FUNCTION_BLOCK Stage11 (* Template for a Basic Function Block Type *)
  (* Standard: 61499-2 *)
  (* Version 1.0, 2021-06-20, HP *)
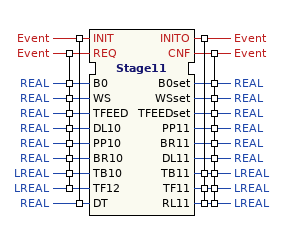
  EVENT_INPUT
    INIT WITH DT; (* Initialization Request *)
    REQ WITH B0, WS, TFEED, DL10, PP10, BR10, TB10, TF12; (* Normal Execution Request *)
  END_EVENT
  EVENT_OUTPUT
    INITO WITH TB11, TF11, RL11; (* Initialization Confirm *)
    CNF WITH PP11, B0set, WSset, TFEEDset, BR11, DL11, TB11, TF11, RL11; (* Execution Confirmation *)
  END_EVENT
  VAR_INPUT
    B0 : REAL;
    WS : REAL;
    TFEED : REAL;
    DL10 : REAL;
    PP10 : REAL;
    BR10 : REAL;
    TB10 : LREAL;
    TF12 : LREAL;
    DT : REAL;
  END_VAR
  VAR_OUTPUT
    B0set : REAL;
    WSset : REAL;
    TFEEDset : REAL;
    PP11 : REAL;
    BR11 : REAL;
    DL11 : REAL;
    TB11 : LREAL;
    TF11 : LREAL;
    RL11 : LREAL;
  END_VAR
  VAR
    AB : REAL; (* internal variabel *)
    UU : REAL;
    TREF : REAL;
    AD : REAL;
    AHC : REAL;
    AHR : REAL;
    AS : REAL;
    REC : REAL;
    WN : REAL;
    WN_1 : REAL;
    XKN : REAL;
    C1 : REAL;
    HS : REAL;
    G : REAL;
    W1 : REAL;
    TFREC : REAL;
    TS : REAL;
    DTS : REAL;
    TF11_last : REAL;
    RL11_last : REAL;
    TB11_last : REAL;
    USS : REAL;
    RHOB : REAL;
    CPB : REAL;
    CPF : REAL;
    FMW : REAL;
    HLV : REAL;
    HV : REAL;
    BPR : REAL;
    FMC : REAL;
    U : REAL;
    A : REAL;
    B : REAL;
    C : REAL;
    D1 : REAL;
    d : REAL;
    a : REAL;
    A1 : REAL;
    A2 : REAL;
    A3 : REAL;
    A4 : REAL;
    A5 : REAL;
    A6 : REAL;
    p : REAL;
    q : REAL;
    TC : REAL;
    PC : REAL;
    DTB11 : REAL;
    DEN11 : REAL;
    DH11 : REAL;
    DP11 : REAL;
    DPDH11 : REAL;
    DT11 : REAL;
    m : REAL;
    n : REAL;
    VR11 : REAL;
    DELTA11 : REAL;
    DELTA33 : REAL;
    DELTA55 : REAL;
    DELTA11_last : REAL;
    DELTA33_last : REAL;
    DELTA55_last : REAL;
  END_VAR
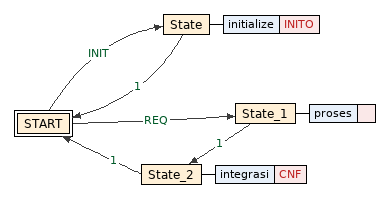
  EC_STATES
    START; (* Initial State *)
    State : initialize -> INITO;
    State_1 : proses;
    State_2 : integrasi -> CNF;
  END_STATES
  EC_TRANSITIONS
    START TO State := INIT;
    State TO START := 1;
    START TO State_1 := REQ;
    State_1 TO State_2 := 1;
    State_2 TO START := 1;
  END_TRANSITIONS
  ALGORITHM initialize IN ST: (* Initialization algorithm *)
TREF :=273.15;
AB :=57.2727;
AHC :=4069.2;
AHR :=2639.7;
AS :=3225.7;
REC :=0.0;
//TF2:=TF2;

//TFEED :=TFEED1+TREF;
 //TS:=TS1+TREF;
WN :=3.0;
XKN :=0.68;
HS:=0.11;
G :=9.81;
W1 :=0.50;

RL11 := 0.579761187999641;
TB11 := 337.917695033442;
TF11 := 334.143160422222;
TF12 := 331.64984152235;


RL11_last :=RL11;
TB11_last :=TB11;
TF11_last :=TF11;
  END_ALGORITHM
  ALGORITHM proses IN ST: (* kalkulasi *)
UU := TFEED;
U :=UU;

USS :=49.767;
C1 :=0.625;
RHOB :=1032.4; //maassa jenis brine
CPB :=1.00; //heatcapacity Brine
CPF :=1.00; //heat capacity feed
FMW :=23654.0;
HLV :=563.7959;
HV :=625.1971;
BPR :=2.192;
FMC :=34736.09;
//U :=UU; //feed temp



///  Calculate the physical properties

//A :=3.2437814;
//B :=5.86826*0.001;
//C :=1.1702379*0.00000001;
//D1 :=2.1878462*0.001;
//TC :=647.27;
//PC :=218.167;


A1 :=3.2437814;
A2:=5.86826*0.001;
A3:=1.1702379*0.00000001;
A4 :=2.1878462*0.001;
A5 :=647.27;
A6 :=218.167;

DTB11 :=A5-TB11;
DEN11 :=(A1+A2*DTB11+A3*DTB11*DTB11*DTB11)/(1+A4*DTB11)*DTB11/TB11;
p:=DEN11;
q:=10.0;
PP11 :=A6/(EXPT(q, p));

// calculate the brine flow rates
DP11:=PP10-PP11;
DH11:=RL11-C1*HS;
DPDH11 :=DP11*101000+G*RHOB*DH11;
m:=DPDH11*RHOB;
n:=0.5;
BR11 :=WN*XKN*RL11*(EXPT(m, n));
BR11 :=BR11*60.0/1000.0;

// calculate the vapor flow rates

DT11 :=TB11-BPR/1.8-(TF12+TF11)*0.5;
VR11:=U*AHC*DT11/HLV/1000.0;
DL11 :=DL10+VR11;


//// state equation
DELTA11 :=(BR10-BR11-VR11)*1000.0/RHOB/AB;
DELTA33 :=((BR10*CPB*(TB10-TB11))-VR11*(HV-CPB*(TB11-TREF)))*1000.0/AB/RHOB/CPB/RL11;
DELTA55 :=(B0*CPF*(TF12-TF11)*1000+(U*AHC*DT11))/FMW/CPF;
  END_ALGORITHM
  ALGORITHM integrasi IN ST: (* new algorithm *)
B0set:=B0;
WSset:=WS ;
TFEEDset:=TFEED;
//integrasi
RL11 := (DELTA11 + DELTA11_last)*0.5*DT + RL11_last;
DELTA11_last :=DELTA11 ;
RL11_last :=RL11;

TB11:= (DELTA33 + DELTA33_last)*0.5*DT + TB11_last;
DELTA33_last :=DELTA33 ;
TB11_last:=TB11;

TF11 := (DELTA55 + DELTA55_last)*0.5*DT + TF11_last;
DELTA55_last :=DELTA55 ;
TF11_last :=TF11;
  END_ALGORITHM
END_FUNCTION_BLOCK
